FUNCTION_BLOCK StationCtrl (* Template for a simple Basic Function Block Type *)
  (* Standard: 61499-2 *)
  (* Version 1.0, 2020-08-10, AK115394 *)
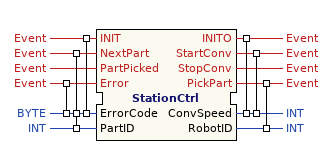
  EVENT_INPUT
    INIT WITH ErrorCode; (* Initialization Request *)
    NextPart WITH PartID, ErrorCode; (* Next part is ready *)
    PartPicked;
    Error WITH ErrorCode; (* Error in system occurred *)
  END_EVENT
  EVENT_OUTPUT
    INITO WITH ConvSpeed; (* Initialization Confirm *)
    StartConv WITH ConvSpeed; (* Execution Confirmation *)
    StopConv;
    PickPart WITH RobotID;
  END_EVENT
  VAR_INPUT
    ErrorCode : BYTE; (* Origin and type of error *)
    PartID : INT;
  END_VAR
  VAR_OUTPUT
    ConvSpeed : INT := 100; (* Output event qualifier *)
    RobotID : INT;
  END_VAR
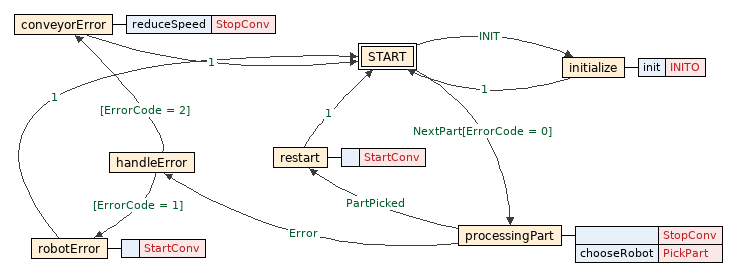
  EC_STATES
    START; (* Initial State *)
    initialize : init -> INITO;
    processingPart : -> StopConv, chooseRobot -> PickPart;
    handleError;
    conveyorError : reduceSpeed -> StopConv;
    robotError : -> StartConv;
    restart : -> StartConv;
  END_STATES
  EC_TRANSITIONS
    START TO initialize := INIT;
    initialize TO START := 1;
    START TO processingPart := NextPart[ErrorCode = 0];
    processingPart TO restart := PartPicked;
    processingPart TO handleError := Error;
    handleError TO robotError := [ErrorCode = 1];
    handleError TO conveyorError := [ErrorCode = 2];
    conveyorError TO START := 1;
    robotError TO START := 1;
    restart TO START := 1;
  END_TRANSITIONS
  ALGORITHM init IN ST: (* Initialization algorithm *)
QO := QI;
  END_ALGORITHM
  ALGORITHM setSpeed IN ST: (* Normally executed algorithm *)
QO := FALSE;
  END_ALGORITHM
  ALGORITHM chooseRobot IN ST: (* new algorithm *)
QO := QI;

IF TRUE  = QI THEN
  (*  only perform normal operation of QI is true*)

END_IF;
  END_ALGORITHM
  ALGORITHM reduceSpeed IN ST:

  END_ALGORITHM
END_FUNCTION_BLOCK
